(* PLC project cam_profile, Dassault Systèmes ControlBuild 2024x *)
(* stored: creationDateTime 2023-10-04T11:03:50-01:00 *)

(* This module is designed to load a cam profile from a file located in "Configuration/camProfiles/" folder of the project *)
FUNCTION_BLOCK motion_lib.cam_profile
  VAR_INPUT
    name : STRING(50) := 'default.txt';
  END_VAR
  VAR_OUTPUT
    nbPoints : INT := 0;
    MasterPoints : ARRAY[1..100] OF REAL := [100(0.0)];
    SlavePoints : ARRAY[1..100] OF REAL := [100(0.0)];
    pointer : DINT := 0;
  END_VAR
  VAR
    initialized : BOOL := false;
    pFile : DINT := 0;
    fault_reading : BOOL := false;
    fault_openning : BOOL := false;
    complete_path : STRING(254) := '';
  END_VAR


ACTION C_source_code:
/* ----------------------------------------------------------------	*/
/* Type : Model of Operative Behaviour					*/
/* Category : motion_control						*/
/* Author : Dassault Systemes						*/
/* Update date : June 2021							*/
/* ----------------------------------------------------------------	*/
/* This module prepares one cam profile tables for the module		*/
/* cam_computation								*/
/* It reads a file made of pair of values :				*/
/* 	<master coord><tab><slave coord>					*/
/* The input file need to be located in the folder 			*/
/* 	/Configuration/camProfiles/						*/
/* of the ControlBuild project						*/
/* ----------------------------------------------------------------	*/

if(!initialized)
{
	initialized = 1;
	fault_openning = 0;
	fault_reading = 0;
	//récupération du chemin complet d'exécution
	GetModuleFileNameA(GetModuleHandle(NULL), projPath, sizeof(projPath));
	for (iPath=0;iPath<6;iPath++) {
		if ((ptrToPathProjet=strrchr(projPath, '\\')) || (ptrToPathProjet=strrchr(projPath, '/')))
			*(ptrToPathProjet) = 0;
	}
	strncpy (completPathToFile, projPath, MAX_PATH);
	strcat(completPathToFile, "/Configuration/camProfiles/");
	completPathToFile[strlen(completPathToFile)] = '\0';

	int inc;
	for(inc=1;inc<=50;inc++){	
		completPathToFile[strlen(completPathToFile)] = name(inc);
	}
	for(inc=1;inc<=254;inc++){	
		complete_path(inc) = completPathToFile[inc-1];
	}

	pFile = fopen(completPathToFile, "r");
	pointer = (camTableStruct*)malloc(sizeof(camTableStruct));
	camTable = pointer;

	if (pFile == 0) {
		fault_openning = 1;
	} else {
		int fin = 0;
		nbPoints = 0;
		while(fin==0) {
			static char str[BUFSIZ];
			char *masterPosC, *slavePosC;
			float masterPos, slavePos;
			if(fgets(str, BUFSIZ, pFile) <= 0) {
				fin = 1;
			} else {
				nbPoints++;
				trim(str);
				if (strlen(str)>1) {
					if (str[strlen(str)-1]=='\n')
						str[strlen(str)-1] = '\0';
					masterPosC = strtok( str, "\t" );
					slavePosC = strtok( NULL, "\t");
					if (slavePosC==NULL || masterPosC==NULL) {
						fault_reading = 1;
					} else {
						sscanf(masterPosC, "%f", &masterPos);
						sscanf(slavePosC, "%f", &slavePos);
						if (nbPoints < 100) {
							MasterPoints(nbPoints) = masterPos;
							SlavePoints(nbPoints) = slavePos;
						}
						camTable->master[nbPoints-1] = masterPos;
						camTable->slave[nbPoints-1] = slavePos;
					}
				}
			}
		}
	}
	initialized = 1;
}
END_ACTION

ACTION C_header:
#include <stdint.h>
#include <sys/time.h>
#include <stdio.h>
#include <stdlib.h>
#include <windows.h>
#include <psapi.h>
#include <shlwapi.h>


char projPath[MAX_PATH];
int iPath;

char* ptrToPathProjet;
char completPathToFile[MAX_PATH];

void trim(char * s) {
    char * p = s;
    int l = strlen(p);

    while(isspace(p[l - 1])) p[--l] = 0;
    while(* p && isspace(* p)) ++p, --l;

    memmove(s, p, l + 1);
}


typedef struct camTableStruct
{  
	float master[7000];
	float slave[7000];
} camTableStruct;

camTableStruct *camTable;
END_ACTION
END_FUNCTION_BLOCK
